PROGRAM Anlage
VAR_INPUT
	UR5				:FB_Roboter;
	Gripper			:FB_SmartGreifer;
	HEX_E			:FB_Kraftsensor; 
END_VAR

VAR
END_VAR

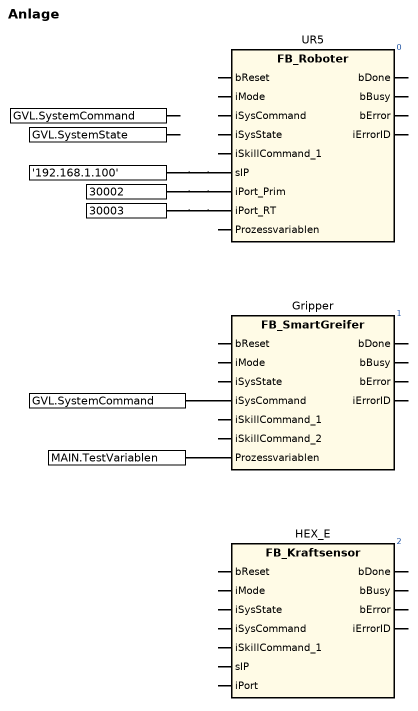
UR5(sIP := '192.168.1.100', iPort_Prim := 30002, iPort_RT := 30003); // FB_Roboter
Gripper(iSysCommand := GVL.SystemCommand, Prozessvariablen := MAIN.TestVariablen); // FB_SmartGreifer
HEX_E(); // FB_Kraftsensor
// GVL.SystemCommand: input not connected
// GVL.SystemState: input not connected

END_PROGRAM

(* stored: Version 1.1.0.1
   POU Anlage: Id {ac0ed22d-45cf-4c60-8691-84647bfee292}, SpecialFunc None *)
